Yaskawa INFORM job: 6.JBI

/JOB
//NAME 6
//POS
///NPOS 14,0,0,0
///TOOL 0
///PULSE
C000=-19991,32580,-29316,-1002,5576,4263
C001=-12551,32580,-29316,-1002,5576,4263
C002=-12607,23928,-28499,-955,5364,4228
C003=-12560,30743,-29395,-1015,5596,4272
C004=-12560,30251,-34874,-2351,6963,5166
C005=-12560,30266,-31944,-1374,6244,4521
C006=-12243,30266,-31940,1249,6245,4105
C007=-12534,30266,-31937,-1153,6246,4486
C008=-12534,30025,-32425,-3206,7343,5824
C009=-12534,30327,-31848,-1029,6029,4402
C010=-11980,30402,-31849,2775,5712,1698
C011=-12534,30327,-31848,-1028,6029,4402
C012=-4970,30329,-31866,-1029,6029,4400
C013=-4970,30329,-31866,-1029,6029,4400
//INST
///DATE 2014/10/13 01:11
///ATTR 0,0,0,0,0,0,0,0,0,0,0,0,0,1,0,0
///FRAME BASE
NOP
MOVJ C000 VJ=0.78 CONT
MOVJ C001 VJ=0.78 CONT
MOVJ C002 VJ=0.78 CONT
MOVJ C003 VJ=0.78 CONT
MOVJ C004 VJ=0.78 CONT
MOVJ C005 VJ=0.78 CONT
MOVJ C006 VJ=0.78 CONT
MOVJ C007 VJ=0.78 CONT
MOVJ C008 VJ=0.78 CONT
MOVJ C009 VJ=0.78 CONT
MOVJ C010 VJ=0.78 CONT
MOVJ C011 VJ=0.78 CONT
MOVJ C012 VJ=0.78 CONT
MOVL C013 V=11.0 CONT
TIMER T=0.01
END
